{attribute 'GeneratedUsingTerminal: EK1960-2600-0021'}
{attribute addProperty BoxType "EK1960-2600-0021"}
{attribute addProperty Id "FSoE_CommandUSINT1FSOUT_Module_1_Channel_1_Output_X5_1BOOL1FSOUT_Module_1_Channel_2_Output_X5_2BOOL1FSOUT_Module_1_Channel_3_Output_X5_3BOOL1FSOUT_Module_1_Channel_4_Output_X5_4BOOL1FSOUT_Module_1_ErrAckBOOL1FSOUT_Module_2_Channel_1_Output_X5_5BOOL1FSOUT_Module_2_Channel_2_Output_X5_6BOOL1FSOUT_Module_2_Channel_3_Output_X5_7BOOL1FSOUT_Module_2_Channel_4_Output_X5_8BOOL1FSOUT_Module_2_ErrAckBOOL1FSOUT_Module_3_Channel_1_Output_X7_1BOOL1FSOUT_Module_3_Channel_2_Output_X7_2BOOL1FSOUT_Module_3_Channel_3_Output_X7_3BOOL1FSOUT_Module_3_Channel_4_Output_X7_4BOOL1FSOUT_Module_3_ErrAckBOOL1FSOUT_Module_4_Channel_1_Output_X7_5BOOL1FSoE_CRC_000UINT2FSOUT_Module_4_Channel_2_Output_X7_6BOOL1FSOUT_Module_4_Channel_3_Output_X7_7BOOL1FSOUT_Module_4_Channel_4_Output_X7_8BOOL1FSOUT_Module_4_ErrAckBOOL1FSOUT_Module_5_Channel_1_Output_X9_1BOOL1FSOUT_Module_5_Channel_2_Output_X9_2BOOL1FSOUT_Module_5_Channel_3_Output_X9_3BOOL1FSOUT_Module_5_Channel_4_Output_X9_4BOOL1FSOUT_Module_5_ErrAckBOOL1FSOUT_Module_6_Channel_1_Output_X9_5BOOL1FSOUT_Module_6_Channel_2_Output_X9_6BOOL1FSOUT_Module_6_Channel_3_Output_X9_7BOOL1FSOUT_Module_6_Channel_4_Output_X9_8BOOL1FSOUT_Module_6_ErrAckBOOL1FSOUT_Relais_Module_Channel_1_Output_X4_1_X4_5BOOL1FSOUT_Relais_Module_Channel_2_Output_X4_2_X4_6BOOL1FSoE_CRC_001UINT2FSOUT_Relais_Module_Channel_3_Output_X4_3_X4_7BOOL1FSOUT_Relais_Module_Channel_4_Output_X4_4_X4_8BOOL1FSOUT_Relais_Module_ErrAckBOOL1FSIN_Module_1_ErrAckBOOL1FSIN_Module_2_ErrAckBOOL1FSIN_Module_3_ErrAckBOOL1FSIN_Module_4_ErrAckBOOL1FSIN_Module_5_ErrAckBOOL1FSIN_Module_6_ErrAckBOOL1FSIN_Module_7_ErrAckBOOL1FSIN_Module_8_ErrAckBOOL1FSIN_Module_9_Err_Ack_1BOOL1FSIN_Module_9_Err_Ack_2BOOL1FSIN_Module_10_Err_Ack_1BOOL1FSIN_Module_10_Err_Ack_2BOOL1FSoE_CRC_002UINT2FSoE_Connection_IDUINT2"}
{attribute addProperty CRC "3455761887"}
{attribute addProperty Size "56"}
TYPE FSOE_CDFABDDF :
STRUCT
	{attribute addProperty Name "FSoE_Command"}
	FSoE_Command : USINT;
	{attribute addProperty Name "FSOUT_Module_1_Channel_1_Output_X5_1"}
	FSOUT_Module_1_Channel_1_Output_X5_1 : BOOL;
	{attribute addProperty Name "FSOUT_Module_1_Channel_2_Output_X5_2"}
	FSOUT_Module_1_Channel_2_Output_X5_2 : BOOL;
	{attribute addProperty Name "FSOUT_Module_1_Channel_3_Output_X5_3"}
	FSOUT_Module_1_Channel_3_Output_X5_3 : BOOL;
	{attribute addProperty Name "FSOUT_Module_1_Channel_4_Output_X5_4"}
	FSOUT_Module_1_Channel_4_Output_X5_4 : BOOL;
	{attribute addProperty Name "FSOUT_Module_1_ErrAck"}
	FSOUT_Module_1_ErrAck : BOOL;
	{attribute addProperty Name "FSOUT_Module_2_Channel_1_Output_X5_5"}
	FSOUT_Module_2_Channel_1_Output_X5_5 : BOOL;
	{attribute addProperty Name "FSOUT_Module_2_Channel_2_Output_X5_6"}
	FSOUT_Module_2_Channel_2_Output_X5_6 : BOOL;
	{attribute addProperty Name "FSOUT_Module_2_Channel_3_Output_X5_7"}
	FSOUT_Module_2_Channel_3_Output_X5_7 : BOOL;
	{attribute addProperty Name "FSOUT_Module_2_Channel_4_Output_X5_8"}
	FSOUT_Module_2_Channel_4_Output_X5_8 : BOOL;
	{attribute addProperty Name "FSOUT_Module_2_ErrAck"}
	FSOUT_Module_2_ErrAck : BOOL;
	{attribute addProperty Name "FSOUT_Module_3_Channel_1_Output_X7_1"}
	FSOUT_Module_3_Channel_1_Output_X7_1 : BOOL;
	{attribute addProperty Name "FSOUT_Module_3_Channel_2_Output_X7_2"}
	FSOUT_Module_3_Channel_2_Output_X7_2 : BOOL;
	{attribute addProperty Name "FSOUT_Module_3_Channel_3_Output_X7_3"}
	FSOUT_Module_3_Channel_3_Output_X7_3 : BOOL;
	{attribute addProperty Name "FSOUT_Module_3_Channel_4_Output_X7_4"}
	FSOUT_Module_3_Channel_4_Output_X7_4 : BOOL;
	{attribute addProperty Name "FSOUT_Module_3_ErrAck"}
	FSOUT_Module_3_ErrAck : BOOL;
	{attribute addProperty Name "FSOUT_Module_4_Channel_1_Output_X7_5"}
	FSOUT_Module_4_Channel_1_Output_X7_5 : BOOL;
	{attribute addProperty Name "FSoE_CRC_000"}
	FSoE_CRC_000 : UINT;
	{attribute addProperty Name "FSOUT_Module_4_Channel_2_Output_X7_6"}
	FSOUT_Module_4_Channel_2_Output_X7_6 : BOOL;
	{attribute addProperty Name "FSOUT_Module_4_Channel_3_Output_X7_7"}
	FSOUT_Module_4_Channel_3_Output_X7_7 : BOOL;
	{attribute addProperty Name "FSOUT_Module_4_Channel_4_Output_X7_8"}
	FSOUT_Module_4_Channel_4_Output_X7_8 : BOOL;
	{attribute addProperty Name "FSOUT_Module_4_ErrAck"}
	FSOUT_Module_4_ErrAck : BOOL;
	{attribute addProperty Name "FSOUT_Module_5_Channel_1_Output_X9_1"}
	FSOUT_Module_5_Channel_1_Output_X9_1 : BOOL;
	{attribute addProperty Name "FSOUT_Module_5_Channel_2_Output_X9_2"}
	FSOUT_Module_5_Channel_2_Output_X9_2 : BOOL;
	{attribute addProperty Name "FSOUT_Module_5_Channel_3_Output_X9_3"}
	FSOUT_Module_5_Channel_3_Output_X9_3 : BOOL;
	{attribute addProperty Name "FSOUT_Module_5_Channel_4_Output_X9_4"}
	FSOUT_Module_5_Channel_4_Output_X9_4 : BOOL;
	{attribute addProperty Name "FSOUT_Module_5_ErrAck"}
	FSOUT_Module_5_ErrAck : BOOL;
	{attribute addProperty Name "FSOUT_Module_6_Channel_1_Output_X9_5"}
	FSOUT_Module_6_Channel_1_Output_X9_5 : BOOL;
	{attribute addProperty Name "FSOUT_Module_6_Channel_2_Output_X9_6"}
	FSOUT_Module_6_Channel_2_Output_X9_6 : BOOL;
	{attribute addProperty Name "FSOUT_Module_6_Channel_3_Output_X9_7"}
	FSOUT_Module_6_Channel_3_Output_X9_7 : BOOL;
	{attribute addProperty Name "FSOUT_Module_6_Channel_4_Output_X9_8"}
	FSOUT_Module_6_Channel_4_Output_X9_8 : BOOL;
	{attribute addProperty Name "FSOUT_Module_6_ErrAck"}
	FSOUT_Module_6_ErrAck : BOOL;
	{attribute addProperty Name "FSOUT_Relais_Module_Channel_1_Output_X4_1_X4_5"}
	FSOUT_Relais_Module_Channel_1_Output_X4_1_X4_5 : BOOL;
	{attribute addProperty Name "FSOUT_Relais_Module_Channel_2_Output_X4_2_X4_6"}
	FSOUT_Relais_Module_Channel_2_Output_X4_2_X4_6 : BOOL;
	{attribute addProperty Name "FSoE_CRC_001"}
	FSoE_CRC_001 : UINT;
	{attribute addProperty Name "FSOUT_Relais_Module_Channel_3_Output_X4_3_X4_7"}
	FSOUT_Relais_Module_Channel_3_Output_X4_3_X4_7 : BOOL;
	{attribute addProperty Name "FSOUT_Relais_Module_Channel_4_Output_X4_4_X4_8"}
	FSOUT_Relais_Module_Channel_4_Output_X4_4_X4_8 : BOOL;
	{attribute addProperty Name "FSOUT_Relais_Module_ErrAck"}
	FSOUT_Relais_Module_ErrAck : BOOL;
	{attribute addProperty Name "FSIN_Module_1_ErrAck"}
	FSIN_Module_1_ErrAck : BOOL;
	{attribute addProperty Name "FSIN_Module_2_ErrAck"}
	FSIN_Module_2_ErrAck : BOOL;
	{attribute addProperty Name "FSIN_Module_3_ErrAck"}
	FSIN_Module_3_ErrAck : BOOL;
	{attribute addProperty Name "FSIN_Module_4_ErrAck"}
	FSIN_Module_4_ErrAck : BOOL;
	{attribute addProperty Name "FSIN_Module_5_ErrAck"}
	FSIN_Module_5_ErrAck : BOOL;
	{attribute addProperty Name "FSIN_Module_6_ErrAck"}
	FSIN_Module_6_ErrAck : BOOL;
	{attribute addProperty Name "FSIN_Module_7_ErrAck"}
	FSIN_Module_7_ErrAck : BOOL;
	{attribute addProperty Name "FSIN_Module_8_ErrAck"}
	FSIN_Module_8_ErrAck : BOOL;
	{attribute addProperty Name "FSIN_Module_9_Err_Ack_1"}
	FSIN_Module_9_Err_Ack_1 : BOOL;
	{attribute addProperty Name "FSIN_Module_9_Err_Ack_2"}
	FSIN_Module_9_Err_Ack_2 : BOOL;
	{attribute addProperty Name "FSIN_Module_10_Err_Ack_1"}
	FSIN_Module_10_Err_Ack_1 : BOOL;
	{attribute addProperty Name "FSIN_Module_10_Err_Ack_2"}
	FSIN_Module_10_Err_Ack_2 : BOOL;
	{attribute addProperty Name "FSoE_CRC_002"}
	FSoE_CRC_002 : UINT;
	{attribute addProperty Name "FSoE_Connection_ID"}
	FSoE_Connection_ID : UINT;
END_STRUCT
END_TYPE

(* stored: Version 1.2.0.0, ProductVersion 3.1.4024.11
   DUT FSOE_CDFABDDF: Id {bab82876-0fae-4c88-a4a0-bcdf9e7add96} *)
